Universal Robots PolyScope program: wrs2020_cable_extend.urp

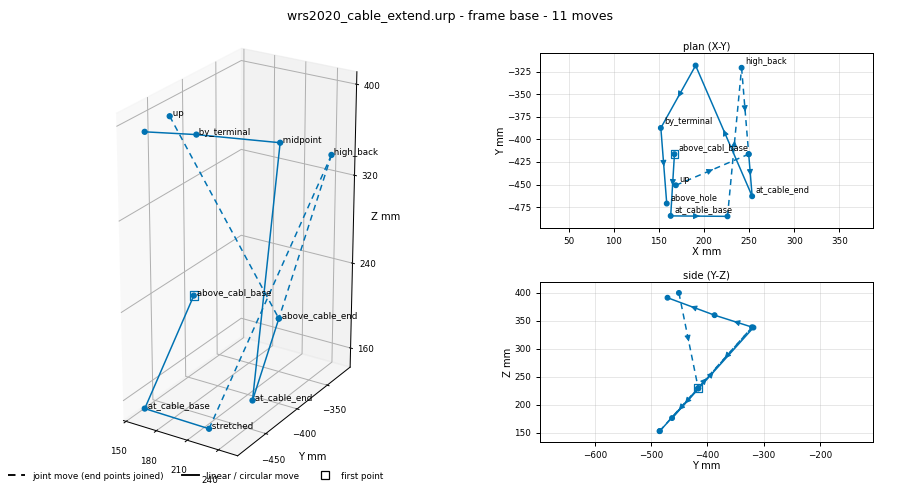
[picture p0: tool path of wrs2020_cable_extend.urp in frame base, 11 of 12 moves have a stored position in this frame; points joined in program order, loops and branches not executed]
Program wrs2020_cable_extend (installation=wrs2020.10 directory=/programs createdIn=5.6.0.90886 lastSavedIn=5.6.0.90886 robotSerialNumber=20205500180)
Calibrated DH parameters: a=[0.000135, -0.030981, -0.334292, 0.000083, 0.000088, 0]; d=[0.162656, 258.79096, -331.603246, 72.945842, 0.099724, 0.099562]; alpha=[1.569535, 0.001639, 0.002824, 1.569633, -1.569323, 0]; deltaTheta=[0, 1.497881, -2.049261, 0.551379, 0, 0]
Robot Program (runOnlyOnce=true)
  URCap Gripper (Robotiq_Grippers, Robotiq Inc.) dataModel(position=71.76470588235294, force=0.0, speed=0.0, positionInDouble=71.76470588235294, forceInDouble=0.0, speedInDouble=0.0, slaveIds=[9], blocking=true)
  MoveL speed 250 mm/s, acceleration 1200 mm/s^2 (useActiveTCP=false) tcp=gripper_140_tip; feature=Base
    Waypoint above_cabl_base: TCP in base x=167.249 y=-416.393 z=229.475 mm, rx=1.8342 ry=-1.8019 rz=0.7367 rad; joints [94.618, -123.285, 140.281, -148.378, -89.759, -86.278] deg; TCP offset x=0 y=0 z=220 mm, rx=0 ry=0 rz=0 rad
    Waypoint at_cable_base: TCP in base x=163.077 y=-484.759 z=153.469 mm, rx=1.7934 ry=-1.8045 rz=0.6719 rad; joints [96.664, -101.667, 141.389, -170.745, -94.78, -84.635] deg
  URCap Gripper (Robotiq_Grippers, Robotiq Inc.) dataModel(position=84.31372549019608, force=0.0, speed=0.0, positionInDouble=84.31372549019608, forceInDouble=0.0, speedInDouble=0.0, slaveIds=[9], blocking=true)
  MoveL speed 250 mm/s, acceleration 1200 mm/s^2 (useActiveTCP=false) tcp=gripper_140_tip; feature=Base
    Waypoint stretched: TCP in base x=226.013 y=-485.267 z=153.158 mm, rx=1.7934 ry=-1.8045 rz=0.6719 rad; joints [107.975, -95.765, 136.479, -170.404, -102.139, -75.917] deg
  Popup Message (haltProgram=false message=wait for b_bot to grasp cable. press enter to move out of the way inputType=Text)
  URCap Gripper (Robotiq_Grippers, Robotiq Inc.) dataModel(position=71.76470588235294, force=0.0, speed=0.0, positionInDouble=71.76470588235294, forceInDouble=0.0, speedInDouble=0.0, slaveIds=[9], blocking=true)
  MoveJ speed 60 deg/s, acceleration 80 deg/s^2 (useActiveTCP=false) tcp=gripper_140_tip; feature=Base
    Waypoint high_back: TCP in base x=241.615 y=-320.675 z=338.164 mm, rx=1.8342 ry=-1.8019 rz=0.7367 rad; joints [121.808, -127.577, 125.129, -125.645, -107.362, -65.273] deg
    Popup Message (haltProgram=false message=wait for b_bot to prepare cable. press enter to pick it inputType=Text)
    Waypoint above_cable_end: TCP in base x=249.492 y=-416.393 z=229.475 mm, rx=1.8342 ry=-1.8019 rz=0.7367 rad; joints [113.089, -111.869, 134.634, -152.634, -101.882, -72.179] deg
  MoveL speed 250 mm/s, acceleration 1200 mm/s^2 (useActiveTCP=false) tcp=gripper_140_tip; feature=Base
    Waypoint at_cable_end: TCP in base x=253.327 y=-463.014 z=176.535 mm, rx=1.8342 ry=-1.8019 rz=0.7367 rad; joints [110.436, -100.303, 136.01, -165.974, -100.199, -74.2] deg
  URCap Gripper (Robotiq_Grippers, Robotiq Inc.) dataModel(position=100.0, force=0.0, speed=0.0, positionInDouble=100.0, forceInDouble=0.0, speedInDouble=0.0, slaveIds=[9], blocking=true)
  Popup Message (haltProgram=false message=press enter, then the robot will regrasp inputType=Text)
  URCap Gripper (Robotiq_Grippers, Robotiq Inc.) dataModel(position=81.96078431372548, force=0.0, speed=0.0, positionInDouble=81.96078431372548, forceInDouble=0.0, speedInDouble=0.0, slaveIds=[9], blocking=true)
  URCap Gripper (Robotiq_Grippers, Robotiq Inc.) dataModel(position=100.0, force=0.0, speed=0.0, positionInDouble=100.0, forceInDouble=0.0, speedInDouble=0.0, slaveIds=[9], blocking=true)
  Popup Message (haltProgram=false message=press enter, then the robot will move to insert inputType=Text)
  MoveL speed 250 mm/s, acceleration 1200 mm/s^2 (useActiveTCP=false) tcp=TCP; feature=Base
    Waypoint midpoint: TCP in base x=190.689 y=-318.186 z=337.618 mm, rx=-0.0483 ry=2.8953 rz=-1.0936 rad; joints [101.131, -105.347, 140.458, -166.296, -94.106, 7.791] deg
    Waypoint by_terminal: TCP in base x=152.165 y=-387.343 z=359.646 mm, rx=-0.0531 ry=2.9653 rz=-0.8939 rad; joints [92.385, -101.917, 131.006, -152.609, -88.17, 0.972] deg
  MoveL speed 250 mm/s, acceleration 1200 mm/s^2 (useActiveTCP=false) tcp=TCP; feature=Base
    Waypoint above_hole: TCP in base x=158.707 y=-471.093 z=390.688 mm, rx=-0.0649 ry=3.0862 rz=-0.332 rad; joints [92.733, -91.899, 109.772, -120.124, -88.039, 0.57] deg
    Popup Message (haltProgram=false message=press enter, then the robot will move to insert inputType=Text)
    Waypoint down (Relative): motionParameters(jointSpeed=1.047198 jointAcceleration=1.396263 cartesianSpeed=0.01 cartesianAcceleration=0.5); relativeFromPosition TCP in base x=169.213 y=-448.693 z=384.09 mm, rx=-0.0649 ry=3.0862 rz=-0.3319 rad; joints [94.252, -94.092, 112.857, -121.052, -88.362, 2.054] deg; TCP in base x=170.384 y=-459.976 z=363.444 mm, rx=-0.0649 ry=3.0862 rz=-0.3318 rad; joints [94.289, -91.461, 113.589, -124.413, -88.369, 2.104] deg
  URCap Gripper (Robotiq_Grippers, Robotiq Inc.) dataModel(position=78.43137254901961, force=0.0, speed=0.0, positionInDouble=78.43137254901961, forceInDouble=0.0, speedInDouble=0.0, slaveIds=[9], blocking=true)
  MoveJ speed 60 deg/s, acceleration 80 deg/s^2 (useActiveTCP=false) tcp=TCP; feature=Base
    Waypoint up: TCP in base x=168.816 y=-450.828 z=399.236 mm, rx=-0.0649 ry=3.0862 rz=-0.332 rad; joints [94.182, -94.491, 110.905, -118.704, -88.349, 1.979] deg
  MoveJ speed 60 deg/s, acceleration 80 deg/s^2 (useActiveTCP=false) tcp=TCP; feature=Base
    Waypoint above_cable_end: TCP in base x=249.492 y=-416.393 z=229.475 mm, rx=1.8342 ry=-1.8019 rz=0.7367 rad; joints [113.089, -111.869, 134.634, -152.634, -101.882, -72.179] deg; TCP offset x=0 y=0 z=220 mm, rx=0 ry=0 rz=0 rad
